TYPE U_WORD :
UNION
	nWORD : WORD;
	st16Bit : ST_16bit;
END_UNION
END_TYPE

(* stored: Version 1.1.0.1, ProductVersion 3.1.4026.6
   DUT U_WORD: Id {dfa93ccf-fe12-46c9-92d2-3aa5ad3e89c8} *)
